{attribute 'qualified_only'}
{attribute 'strict'}
{attribute 'to_string'}
TYPE ST125_Pnp_e :
(
    RESET := 0, // Reset

    INIT := 100, // Initialisieren 
    Init_HomeVerticals,
    Init_VerticalsUp,
	Init_open_solenohr_gripper,
	Init_handling_up,
    Init_HomeHorizontals,
    Init_HorizontalsToTrack,
	Init_check_if_pces_handled,

    READY := 999,  // READY to Start, Init Done 
    START := 1000, // Start Zyklisch
    MOVER_FREE_OP, // Ab here, operation without mover can be done

    Pnp_Hor_ToRotTablePos,
    Pnp_WaitOnFeeder,
    Pnp_Ver_RotTableDown,
    Pnp_takeTubeCap,
    Pnp_Ver_RotTableUp,
    Pnp_Hor_ToTrackPos,
    waitOnMover,     // wait until the mover is there
    MOVER_NEEDED_OP, // Since here, a mover in position is needed to perform the action

    Pnp_HandlingDown,
    Pnp_Ver_ShuttleDown,
    Pnp_HandlingSolerohrMaintain,
    Pnp_Ver_ShuttleTorqueControl,
    Pnp_putTubeCap,
    Pnp_Ver_ShuttleUpToHandling,
    Pnp_HandlingSolerohrRelease,
    Pnp_Ver_ShuttleFullUp,
    Pnp_HandlingUp,

    SYNC_MOVER_LEAVE, // MoverMan need to take the mover
    DONE := 8000,     // Ablauf beendet 
    ERROR := 9000,    // Fehler 
    _max
);
END_TYPE

(* stored: Version 1.1.0.1, ProductVersion 3.1.4024.6
   EnumerationTextList ST125_Pnp_e: Id {11dccf01-1e1e-4f86-95b3-a5c4ef7fc123} *)
